Staubli VAL3: saveIt.pgx

program saveIt(bool& x_bSave[])
  local string l_sMessage
  local num l_nResult
  local num l_nType
  local string l_sPath
begin
  // unselect ALL
  call prog:unSelectItem()
  // save
  call prog:save(sProgram,l_nResult)
  if l_nResult==0
    logMsg("[KERNEL] INTERFACE:Save the program: "+sProgram)
    x_bSave=false
    call language:message(l_sMessage,-4)
    call use:timerDialog(l_sMessage,1)
  else
    popUpMsg("Save code error "+toString("",l_nResult))
  endIf
end
